{attribute 'qualified_only'}
{attribute 'strict'}
TYPE eVFD :
(
	IN_RUN_STOP := 14,
	IN_SPEED_1	:= 15,
	IN_SPEED_2	:= 16,
	OUT_READY 	:= 20,
	OUT_24		:= 24,
	OUT_26		:= 26
	
);
END_TYPE

(* stored: Version 1.1.0.1, ProductVersion 3.1.4024.10
   EnumerationTextList eVFD: Id {8340ea3b-a06a-421a-a8f9-6cf587ed3f6d} *)
